(******************************************************************************
Baustein: FB_UnitTestBase
Spezifikation: doc/Spezifikation.pdf, Kap. x.y.z
-------------------------------------------------------------------------------
erstellt:
von:
Geändert:
von:
-------------------------------------------------------------------------------
Beschreibung
Dieser Baustein stellt die Basis für einen Unittest dar und enthält
alle notwendigen Variablen und Methoden zur Testauswertung.

-------------------------------------------------------------------------------
Input
-

Output
	o_eState : EState_t;
	o_eResult: EResult_t;
******************************************************************************)
FUNCTION_BLOCK FB_UnitTestBase
VAR_INPUT
END_VAR
VAR_OUTPUT
	o_eState : EState_t;
	o_eResult: EResult_t;
END_VAR
VAR
	strId	  		: ObjectId_t;
	strClassName	: ObjectId_t;
	strPath			: ObjectId_t;
	strMessage 	 	: StrMessage_t;
	bSkipTest		: BOOL;
	pTestSuite      : TestSuiteHandle_t;
	bRegistered 	: BOOL;
	u32Passed 		: UDINT;
	u32Failed 		: UDINT;
	u32StartTime	: UDINT;
	u32EndTime		: UDINT;
END_VAR

(******************************************************************************
Baustein: FB_UnitTestBase.cleanup
Spezifikation: doc/Spezifikation.pdf, Kap. x.y.z
-------------------------------------------------------------------------------
erstellt:
von:
Geändert:
von:
-------------------------------------------------------------------------------
Beschreibung
Diese Methode...

-------------------------------------------------------------------------------
Input
-

Output
-
******************************************************************************)
{attribute 'hide'} 
METHOD INTERNAL _cleanup : BOOL
VAR_INPUT
END_VAR


	_cleanup := cleanup();
END_METHOD

(******************************************************************************
Baustein: FB_UnitTestBase.execute
Spezifikation: doc/Spezifikation.pdf, Kap. x.y.z
-------------------------------------------------------------------------------
erstellt:
von:
Geändert:
von:
-------------------------------------------------------------------------------
Beschreibung
Diese Methode...

-------------------------------------------------------------------------------
Input
-

Output
-
******************************************************************************)
{attribute 'hide'} 
METHOD INTERNAL _execute : BOOL
VAR_INPUT
END_VAR

	_execute := execute();
END_METHOD

(******************************************************************************
Baustein: FB_UnitTestBase.prepare
Spezifikation: doc/Spezifikation.pdf, Kap. x.y.z
-------------------------------------------------------------------------------
erstellt:
von:
Geändert:
von:
-------------------------------------------------------------------------------
Beschreibung
Diese Methode...

-------------------------------------------------------------------------------
Input
-

Output
-
******************************************************************************)
{attribute 'hide'} 
METHOD INTERNAL _prepare : BOOL
VAR_INPUT
END_VAR

	u32Passed 		:= 0;
	u32Failed 		:= 0;
	u32StartTime 	:= 0;
	u32EndTime 		:= 0;
	o_eResult 		:= EResult_t.eStateSkipped;

	_prepare := prepare();
END_METHOD

(******************************************************************************
Baustein: FB_UnitTestBase.addFailed
Spezifikation: doc/Spezifikation.pdf, Kap. x.y.z
-------------------------------------------------------------------------------
erstellt:
von:
Geändert:
von:
-------------------------------------------------------------------------------
Beschreibung
Diese Methode

-------------------------------------------------------------------------------
Input
-

Output
-
******************************************************************************)
{attribute 'hide'} 
METHOD INTERNAL addFailed : BOOL
VAR_INPUT
	bFatal : BOOL;
END_VAR

	u32Failed := u32Failed + 1;
	
	o_eResult := EResult_t.eStateFailed;
	
	IF bFatal = true THEN
		o_eResult := EResult_t.eStateFailedFatal;
		logError(concat('Test Failed Fatal: ', strId));
	ELSE
		logError(concat('Test Failed : ', strId));
	END_IF
END_METHOD

(******************************************************************************
Baustein: FB_UnitTestBase.addPassed
Spezifikation: doc/Spezifikation.pdf, Kap. x.y.z
-------------------------------------------------------------------------------
erstellt:
von:
Geändert:
von:
-------------------------------------------------------------------------------
Beschreibung
Diese Methode

-------------------------------------------------------------------------------
Input
-

Output
-
******************************************************************************)
{attribute 'hide'} 
METHOD INTERNAL addPassed : BOOL
VAR_INPUT
END_VAR

	u32Passed := u32Passed + 1;

	IF o_eResult = eResult_t.eStateSkipped THEN
		o_eResult := eResult_t.eStatePassed;
	END_IF;
END_METHOD

(******************************************************************************
Baustein: FB_UnitTestBase.assertEQUAL
Spezifikation: doc/Spezifikation.pdf, Kap. x.y.z
-------------------------------------------------------------------------------
erstellt:
von:
Geändert:
von:
-------------------------------------------------------------------------------
Beschreibung
Diese Methode

-------------------------------------------------------------------------------
Input
	Actual   : ANY;
	Expected : ANY;

Output
-
******************************************************************************)
METHOD PROTECTED assertEQUAL : BOOL
VAR_INPUT
	Actual   : ANY;
	Expected : ANY;
END_VAR

	assertEQUAL := FALSE;
	
	IF validate(Actual, Expected) = FALSE THEN
		addFailed(true);
		RETURN;
	END_IF
	
	assertTrue(MEMCMP(Actual.pValue, Expected.pValue, TO_UDINT(Actual.diSize)) = 0);
END_METHOD

(******************************************************************************
Baustein: FB_UnitTestBase.assertEQUAL_Fatal
Spezifikation: doc/Spezifikation.pdf, Kap. x.y.z
-------------------------------------------------------------------------------
erstellt:
von:
Geändert:
von:
-------------------------------------------------------------------------------
Beschreibung
Diese Methode

-------------------------------------------------------------------------------
Input
	Actual   : ANY;
	Expected : ANY;

Output
-
******************************************************************************)
METHOD PROTECTED assertEQUAL_Fatal : BOOL
VAR_INPUT
	Actual   : ANY;
	Expected : ANY;
END_VAR

	assertEQUAL_Fatal := FALSE;
	
	IF validate(Actual, Expected) = FALSE THEN
		addFailed(true);
		RETURN;
	END_IF

	assertTrue_Fatal(MEMCMP(Actual.pValue, Expected.pValue, TO_UDINT(Actual.diSize)) = 0);
END_METHOD

(******************************************************************************
Baustein: FB_UnitTestBase.assertFALSE
Spezifikation: doc/Spezifikation.pdf, Kap. x.y.z
-------------------------------------------------------------------------------
erstellt:
von:
Geändert:
von:
-------------------------------------------------------------------------------
Beschreibung
Diese Methode...

-------------------------------------------------------------------------------
Input
	bValue : BOOL;

Output
-
******************************************************************************)
METHOD PROTECTED assertFALSE : BOOL
VAR_INPUT
	bValue : BOOL;
END_VAR

	IF bValue = FALSE THEN
		addPassed();
	ELSE
		addFailed(bFatal := FALSE);
	END_IF
END_METHOD

(******************************************************************************
Baustein: FB_UnitTestBase.assertFALSE_Fatal
Spezifikation: doc/Spezifikation.pdf, Kap. x.y.z
-------------------------------------------------------------------------------
erstellt:
von:
Geändert:
von:
-------------------------------------------------------------------------------
Beschreibung
Diese Methode

-------------------------------------------------------------------------------
Input
	bValue : BOOL;

Output
-
******************************************************************************)
METHOD PROTECTED assertFALSE_Fatal : BOOL
VAR_INPUT
	bValue : BOOL;
END_VAR

	IF bValue = FALSE THEN
		addPassed();
	ELSE
		addFailed(bFatal := true);
	END_IF
END_METHOD

(******************************************************************************
Baustein: FB_UnitTestBase.assertNotEqual
Spezifikation: doc/Spezifikation.pdf, Kap. x.y.z
-------------------------------------------------------------------------------
erstellt:
von:
Geändert:
von:
-------------------------------------------------------------------------------
Beschreibung
Diese Methode

-------------------------------------------------------------------------------
Input
	Actual   : ANY;
	Expected : ANY;

Output
-
******************************************************************************)
METHOD PROTECTED assertNotEqual : BOOL
VAR_INPUT
	Actual   : ANY;
	Expected : ANY;
END_VAR

	assertNotEqual := FALSE;
	
	IF validate(Actual, Expected) = FALSE THEN
		addFailed(true);
		RETURN;
	END_IF
	
	assertTrue(MEMCMP(Actual.pValue, Expected.pValue, TO_UDINT(Actual.diSize)) <> 0);
END_METHOD

(******************************************************************************
Baustein: FB_UnitTestBase.assertNotEqual_Fatal
Spezifikation: doc/Spezifikation.pdf, Kap. x.y.z
-------------------------------------------------------------------------------
erstellt:
von:
Geändert:
von:
-------------------------------------------------------------------------------
Beschreibung
Diese Methode

-------------------------------------------------------------------------------
Input
	Actual   : ANY;
	Expected : ANY;

Output
-
******************************************************************************)
METHOD PROTECTED assertNotEqual_Fatal : BOOL
VAR_INPUT
	Actual   : ANY;
	Expected : ANY;
END_VAR

	assertNotEqual_Fatal := FALSE;
	
	IF validate(Actual, Expected) = FALSE THEN
		addFailed(true);
		RETURN;
	END_IF
	
	assertTrue_Fatal(MEMCMP(Actual.pValue, Expected.pValue, TO_UDINT(Actual.diSize)) <> 0);
END_METHOD

(******************************************************************************
Baustein: FB_UnitTestBase.assertPtrEqual
Spezifikation: doc/Spezifikation.pdf, Kap. x.y.z
-------------------------------------------------------------------------------
erstellt:
von:
Geändert:
von:
-------------------------------------------------------------------------------
Beschreibung
Diese Methode

-------------------------------------------------------------------------------
Input
	pActual   : PVOID;
	pExpected : PVOID;
	
Output
-
******************************************************************************)
METHOD PROTECTED assertPtrEqual : BOOL
VAR_INPUT
	pActual   : PVOID;
	pExpected : PVOID;
END_VAR

	assertTRUE(pActual = pExpected);
END_METHOD

(******************************************************************************
Baustein: FB_UnitTestBase.assertPtrEqual_Fatal
Spezifikation: doc/Spezifikation.pdf, Kap. x.y.z
-------------------------------------------------------------------------------
erstellt:
von:
Geändert:
von:
-------------------------------------------------------------------------------
Beschreibung
Diese Methode

-------------------------------------------------------------------------------
Input
	pActual   : PVOID;
	pExpected : PVOID;

Output
-
******************************************************************************)
METHOD PROTECTED assertPtrEqual_Fatal : BOOL
VAR_INPUT
	pActual   : PVOID;
	pExpected : PVOID;
END_VAR

	assertTRUE_Fatal(pActual = pExpected);
END_METHOD

(******************************************************************************
Baustein: FB_UnitTestBase.assertPtrNotEqual
Spezifikation: doc/Spezifikation.pdf, Kap. x.y.z
-------------------------------------------------------------------------------
erstellt:
von:
Geändert:
von:
-------------------------------------------------------------------------------
Beschreibung
Diese Methode

-------------------------------------------------------------------------------
Input
	pActual   : PVOID;
	pExpected : PVOID;

Output
-
******************************************************************************)
METHOD PROTECTED assertPtrNotEqual : BOOL
VAR_INPUT
	pActual   : PVOID;
	pExpected : PVOID;
END_VAR

	assertTRUE(pActual <> pExpected);
END_METHOD

(******************************************************************************
Baustein: FB_UnitTestBase.assertPtrNotEqual_Fatal
Spezifikation: doc/Spezifikation.pdf, Kap. x.y.z
-------------------------------------------------------------------------------
erstellt:
von:
Geändert:
von:
-------------------------------------------------------------------------------
Beschreibung
Diese Methode

-------------------------------------------------------------------------------
Input
	pActual   : PVOID;
	pExpected : PVOID;

Output
-
******************************************************************************)
METHOD PROTECTED assertPtrNotEqual_Fatal : BOOL
VAR_INPUT
	pActual   : PVOID;
	pExpected : PVOID;
END_VAR

	assertTRUE_Fatal(pActual <> pExpected);
END_METHOD

(******************************************************************************
Baustein: FB_UnitTestBase.assertPtrNotNull
Spezifikation: doc/Spezifikation.pdf, Kap. x.y.z
-------------------------------------------------------------------------------
erstellt:
von:
Geändert:
von:
-------------------------------------------------------------------------------
Beschreibung
Diese Methode

-------------------------------------------------------------------------------
Input
	pActual   : PVOID;

Output
-
******************************************************************************)
METHOD PROTECTED assertPtrNotNull : BOOL
VAR_INPUT
	pActual   : PVOID;
END_VAR

	assertTRUE(pActual <> 0);
END_METHOD

(******************************************************************************
Baustein: FB_UnitTestBase.assertPtrNotNull_Fatal
Spezifikation: doc/Spezifikation.pdf, Kap. x.y.z
-------------------------------------------------------------------------------
erstellt:
von:
Geändert:
von:
-------------------------------------------------------------------------------
Beschreibung
Diese Methode

-------------------------------------------------------------------------------
Input
	pActual   : PVOID;

Output
-
******************************************************************************)
METHOD PROTECTED assertPtrNotNull_Fatal : BOOL
VAR_INPUT
	pActual   : PVOID;
END_VAR

	assertTRUE_Fatal(pActual <> 0);
END_METHOD

(******************************************************************************
Baustein: FB_UnitTestBase.assertPtrNull
Spezifikation: doc/Spezifikation.pdf, Kap. x.y.z
-------------------------------------------------------------------------------
erstellt:
von:
Geändert:
von:
-------------------------------------------------------------------------------
Beschreibung
Diese Methode

-------------------------------------------------------------------------------
Input
	pActual   : PVOID;

Output
-
******************************************************************************)
METHOD PROTECTED assertPtrNull : BOOL
VAR_INPUT
	pActual   : PVOID;
END_VAR

	assertTRUE(pActual = 0);
END_METHOD

(******************************************************************************
Baustein: FB_UnitTestBase.assertPtrNull_Fatal
Spezifikation: doc/Spezifikation.pdf, Kap. x.y.z
-------------------------------------------------------------------------------
erstellt:
von:
Geändert:
von:
-------------------------------------------------------------------------------
Beschreibung
Diese Methode

-------------------------------------------------------------------------------
Input
	pActual   : PVOID;

Output
-
******************************************************************************)
METHOD PROTECTED assertPtrNull_Fatal : BOOL
VAR_INPUT
	pActual   : PVOID;
END_VAR

	assertTRUE_Fatal(pActual = 0);
END_METHOD

(******************************************************************************
Baustein: FB_UnitTestBase.assertRealEqual
Spezifikation: doc/Spezifikation.pdf, Kap. x.y.z
-------------------------------------------------------------------------------
erstellt:
von:
Geändert:
von:
-------------------------------------------------------------------------------
Beschreibung
Diese Methode

-------------------------------------------------------------------------------
Input
	r32Actual 		: REAL;
	r32Expected 	: REAL;
	r32Granularity 	: REAL;

Output
-
******************************************************************************)
METHOD PROTECTED assertRealEqual : BOOL
VAR_INPUT
	r32Actual 		: REAL;
	r32Expected 	: REAL;
	r32Granularity 	: REAL;
END_VAR

	assertTRUE(ABS(r32Actual-r32Expected) <= ABS(r32Granularity));
END_METHOD

(******************************************************************************
Baustein: FB_UnitTestBase.assertRealEqual_Fatal
Spezifikation: doc/Spezifikation.pdf, Kap. x.y.z
-------------------------------------------------------------------------------
erstellt:
von:
Geändert:
von:
-------------------------------------------------------------------------------
Beschreibung
Diese Methode

-------------------------------------------------------------------------------
Input
	r32Actual 		: REAL;
	r32Expected 	: REAL;
	r32Granularity 	: REAL;

Output
-
******************************************************************************)
METHOD PROTECTED assertRealEqual_Fatal : BOOL
VAR_INPUT
	r32Actual 		: REAL;
	r32Expected 	: REAL;
	r32Granularity 	: REAL;
END_VAR

	assertTRUE_Fatal(ABS(r32Actual-r32Expected) <= ABS(r32Granularity));
END_METHOD

(******************************************************************************
Baustein: FB_UnitTestBase.assertRealNotEqual
Spezifikation: doc/Spezifikation.pdf, Kap. x.y.z
-------------------------------------------------------------------------------
erstellt:
von:
Geändert:
von:
-------------------------------------------------------------------------------
Beschreibung
Diese Methode

-------------------------------------------------------------------------------
Input
	r32Actual 		: REAL;
	r32Expected 	: REAL;
	r32Granularity 	: REAL;

Output
-
******************************************************************************)
METHOD PRIVATE assertRealNotEqual : BOOL
VAR_INPUT
	r32Actual 		: REAL;
	r32Expected 	: REAL;
	r32Granularity 	: REAL;
END_VAR

	assertTRUE(ABS(r32Actual-r32Expected) > ABS(r32Granularity));
END_METHOD

(******************************************************************************
Baustein: FB_UnitTestBase.assertRealNotEqual_Fatal
Spezifikation: doc/Spezifikation.pdf, Kap. x.y.z
-------------------------------------------------------------------------------
erstellt:
von:
Geändert:
von:
-------------------------------------------------------------------------------
Beschreibung
Diese Methode

-------------------------------------------------------------------------------
Input
	r32Actual 		: REAL;
	r32Expected 	: REAL;
	r32Granularity 	: REAL;

Output
-
******************************************************************************)
METHOD PROTECTED assertRealNotEqual_Fatal : BOOL
VAR_INPUT
	r32Actual 		: REAL;
	r32Expected 	: REAL;
	r32Granularity 	: REAL;
END_VAR

	assertTRUE_Fatal(ABS(r32Actual-r32Expected) > ABS(r32Granularity));
END_METHOD

(******************************************************************************
Baustein: FB_UnitTestBase.assertStringEqual
Spezifikation: doc/Spezifikation.pdf, Kap. x.y.z
-------------------------------------------------------------------------------
erstellt:
von:
Geändert:
von:
-------------------------------------------------------------------------------
Beschreibung
Diese Methode

-------------------------------------------------------------------------------
Input
	pActual 	: StringHandle_t;
	pExpected 	: StringHandle_t;

Output
-
******************************************************************************)
METHOD PROTECTED assertStringEqual : BOOL
VAR_INPUT
	pActual 	: StringHandle_t;
	pExpected 	: StringHandle_t;
END_VAR

	IF strncmp(pActual, pExpected, LEN(pExpected^)) = TRUE THEN
		addPassed();
	ELSE
		addFailed(bFatal := FALSE);		
	END_IF
END_METHOD

(******************************************************************************
Baustein: FB_UnitTestBase.assertStringEqual_Fatal
Spezifikation: doc/Spezifikation.pdf, Kap. x.y.z
-------------------------------------------------------------------------------
erstellt:
von:
Geändert:
von:
-------------------------------------------------------------------------------
Beschreibung
Diese Methode

-------------------------------------------------------------------------------
Input
	pActual 	: StringHandle_t;
	pExpected 	: StringHandle_t;

Output
-
******************************************************************************)
METHOD PROTECTED assertStringEqual_Fatal : BOOL
VAR_INPUT
	pActual 	: StringHandle_t;
	pExpected 	: StringHandle_t;
END_VAR

	IF strncmp(pActual, pExpected, LEN(pExpected^)) = TRUE THEN
		addPassed();
	ELSE
		addFailed(bFatal := TRUE);		
	END_IF
END_METHOD

(******************************************************************************
Baustein: FB_UnitTestBase.assertStringNotEqual
Spezifikation: doc/Spezifikation.pdf, Kap. x.y.z
-------------------------------------------------------------------------------
erstellt:
von:
Geändert:
von:
-------------------------------------------------------------------------------
Beschreibung
Diese Methode

-------------------------------------------------------------------------------
Input
	pActual 	: StringHandle_t;
	pExpected 	: StringHandle_t;

Output
-
******************************************************************************)
METHOD PROTECTED assertStringNotEqual : BOOL
VAR_INPUT
	pActual 	: StringHandle_t;
	pExpected 	: StringHandle_t;
END_VAR

	IF strncmp(pActual, pExpected, LEN(pExpected^)) = false THEN
		addPassed();
	ELSE
		addFailed(bFatal := FALSE);		
	END_IF
END_METHOD

(******************************************************************************
Baustein: FB_UnitTestBase.assertStringNotEqual_fatal
Spezifikation: doc/Spezifikation.pdf, Kap. x.y.z
-------------------------------------------------------------------------------
erstellt:
von:
Geändert:
von:
-------------------------------------------------------------------------------
Beschreibung
Diese Methode

-------------------------------------------------------------------------------
Input
	pExpected 	: StringHandle_t;
	pActual 	: StringHandle_t;

Output
-
******************************************************************************)
METHOD PROTECTED assertStringNotEqual_fatal : BOOL
VAR_INPUT
	pExpected 	: StringHandle_t;
	pActual 	: StringHandle_t;
END_VAR

	IF strncmp(pActual, pExpected, LEN(pExpected^)) = FALSE THEN
		addPassed();
	ELSE
		addFailed(bFatal := TRUE);		
	END_IF
END_METHOD

(******************************************************************************
Baustein: FB_UnitTestBase.assertTRUE
Spezifikation: doc/Spezifikation.pdf, Kap. x.y.z
-------------------------------------------------------------------------------
erstellt:
von:
Geändert:
von:
-------------------------------------------------------------------------------
Beschreibung
Diese Methode...

-------------------------------------------------------------------------------
Input
	bValue : BOOL;

Output
-
******************************************************************************)
METHOD PROTECTED assertTRUE : BOOL
VAR_INPUT
	bValue : BOOL;
END_VAR

	IF bValue = true THEN
		addPassed();
	ELSE
		addFailed(bFatal := FALSE);
	END_IF
END_METHOD


(******************************************************************************
Baustein: FB_UnitTestBase.assertTRUE_Fatal
Spezifikation: doc/Spezifikation.pdf, Kap. x.y.z
-------------------------------------------------------------------------------
erstellt:
von:
Geändert:
von:
-------------------------------------------------------------------------------
Beschreibung
Diese Methode

-------------------------------------------------------------------------------
Input
-

Output
-
******************************************************************************)
METHOD PROTECTED assertTRUE_Fatal : BOOL
VAR_INPUT
	bValue : BOOL;
END_VAR

	IF bValue = TRUE THEN
		addPassed();
	ELSE
		addFailed(bFatal := true);
	END_IF
END_METHOD

(******************************************************************************
Baustein: FB_UnitTestBase.cleanup
Spezifikation: doc/Spezifikation.pdf, Kap. x.y.z
-------------------------------------------------------------------------------
erstellt:
von:
Geändert:
von:
-------------------------------------------------------------------------------
Beschreibung
Diese Methode...

-------------------------------------------------------------------------------
Input
-

Output
-
******************************************************************************)
METHOD PUBLIC cleanup : BOOL
VAR_INPUT
END_VAR


	cleanup := false;
END_METHOD

(******************************************************************************
Baustein: FB_UnitTestBase.execute
Spezifikation: doc/Spezifikation.pdf, Kap. x.y.z
-------------------------------------------------------------------------------
erstellt:
von:
Geändert:
von:
-------------------------------------------------------------------------------
Beschreibung
Diese Methode...

-------------------------------------------------------------------------------
Input
-

Output
-
******************************************************************************)
METHOD PUBLIC execute : BOOL
VAR_INPUT
END_VAR

	Execute := false;
END_METHOD

(******************************************************************************
Baustein: FB_Testsuite.FB_init
Spezifikation: doc/Spezifikation.pdf, Kap. x.y.z
-------------------------------------------------------------------------------
erstellt:
von:
Geändert:
von:
-------------------------------------------------------------------------------
Beschreibung
Diese Methode

-------------------------------------------------------------------------------
Input
-

Output
-
******************************************************************************)
{attribute 'hide'} 
METHOD FB_init : BOOL
VAR_INPUT
	bInitRetains 	: BOOL; // if TRUE, the retain variables are initialized (warm start / cold start)
	bInCopyCode 	: BOOL;  // if TRUE, the instance afterwards gets moved into the copy code (online change)
	i_strId	  		: ObjectId_t;
	i_strClassName	: ObjectId_t;
	i_strPath 		: ObjectId_t;
	i_pTestSuite 	: TestSuiteHandle_t;
	i_bExecute      : BOOL := true; 
END_VAR
	
	strId 		 := i_strId;
	strClassName := i_strClassName;
	strPath 	 := i_strPath;
	bSkipTest  	 := (i_bExecute = false);
	pTestSuite 	 := i_pTestSuite;
	
	register();
END_METHOD

(******************************************************************************
Baustein: FB_UnitTestBase.getId
Spezifikation: doc/Spezifikation.pdf, Kap. x.y.z
-------------------------------------------------------------------------------
erstellt:
von:
Geändert:
von:
-------------------------------------------------------------------------------
Beschreibung
Diese Methode

-------------------------------------------------------------------------------
Input
-

Output
-
******************************************************************************)
{attribute 'hide'} 
METHOD PUBLIC getClassName : ObjectId_t
VAR_INPUT
END_VAR

	getClassName := strClassName;
END_METHOD

(******************************************************************************
Baustein: FB_UnitTestBase.getFailed
Spezifikation: doc/Spezifikation.pdf, Kap. x.y.z
-------------------------------------------------------------------------------
erstellt:
von:
Geändert:
von:
-------------------------------------------------------------------------------
Beschreibung
Diese Methode

-------------------------------------------------------------------------------
Input
-

Output
-
******************************************************************************)
{attribute 'hide'} 
METHOD PUBLIC getFailed : UDINT
VAR_INPUT
END_VAR

	getFailed := u32Failed;
END_METHOD

(******************************************************************************
Baustein: FB_UnitTestBase.getId
Spezifikation: doc/Spezifikation.pdf, Kap. x.y.z
-------------------------------------------------------------------------------
erstellt:
von:
Geändert:
von:
-------------------------------------------------------------------------------
Beschreibung
Diese Methode

-------------------------------------------------------------------------------
Input
-

Output
-
******************************************************************************)
{attribute 'hide'} 
METHOD PUBLIC getId : ObjectId_t
VAR_INPUT
END_VAR

	getId := strId;
END_METHOD

METHOD PUBLIC getMessage : StrMessage_t
VAR_INPUT
END_VAR

	getMessage := strMessage;
END_METHOD

(******************************************************************************
Baustein: FB_UnitTestBase.getPassed
Spezifikation: doc/Spezifikation.pdf, Kap. x.y.z
-------------------------------------------------------------------------------
erstellt:
von:
Geändert:
von:
-------------------------------------------------------------------------------
Beschreibung
Diese Methode

-------------------------------------------------------------------------------
Input
-

Output
-
******************************************************************************)
{attribute 'hide'} 
METHOD PUBLIC getPassed : UDINT
VAR_INPUT
END_VAR

	getPassed := u32Passed;
END_METHOD

(******************************************************************************
Baustein: FB_UnitTestBase.getPassed
Spezifikation: doc/Spezifikation.pdf, Kap. x.y.z
-------------------------------------------------------------------------------
erstellt:
von:
Geändert:
von:
-------------------------------------------------------------------------------
Beschreibung
Diese Methode

-------------------------------------------------------------------------------
Input
-

Output
-
******************************************************************************)
{attribute 'hide'} 
METHOD PUBLIC getPath : ObjectId_t
VAR_INPUT
END_VAR

	getPath := strPath;
END_METHOD

(******************************************************************************
Baustein: FB_UnitTestBase.getPassed
Spezifikation: doc/Spezifikation.pdf, Kap. x.y.z
-------------------------------------------------------------------------------
erstellt:
von:
Geändert:
von:
-------------------------------------------------------------------------------
Beschreibung
Diese Methode

-------------------------------------------------------------------------------
Input
-

Output
-
******************************************************************************)
{attribute 'hide'} 
METHOD PRIVATE getSystemTime : UDINT
VAR_INPUT
END_VAR
VAR
	u64Time : ULINT;
END_VAR

	u64Time := F_GetSystemTime()/10000;


	getSystemTime := to_udint(u64Time and 16#FFFFFFFF);
END_METHOD

(******************************************************************************
Baustein: FB_UnitTestBase.getPassed
Spezifikation: doc/Spezifikation.pdf, Kap. x.y.z
-------------------------------------------------------------------------------
erstellt:
von:
Geändert:
von:
-------------------------------------------------------------------------------
Beschreibung
Diese Methode

-------------------------------------------------------------------------------
Input
-

Output
-
******************************************************************************)
{attribute 'hide'} 
METHOD PUBLIC getTime : UDINT
VAR_INPUT
END_VAR

	getTime := 0;

	IF u32EndTime > u32StartTime THEN
		getTime := u32EndTime - u32StartTime;
	END_IF;
END_METHOD

(******************************************************************************
Baustein: FB_UnitTestBase.getPassed
Spezifikation: doc/Spezifikation.pdf, Kap. x.y.z
-------------------------------------------------------------------------------
erstellt:
von:
Geändert:
von:
-------------------------------------------------------------------------------
Beschreibung
Diese Methode

-------------------------------------------------------------------------------
Input
-

Output
-
******************************************************************************)
{attribute 'hide'} 
METHOD INTERNAL isSkipped : BOOL
VAR_INPUT
END_VAR

	isSkipped := bSkipTest;
END_METHOD

(******************************************************************************
Baustein: FB_UnitTestBase.logError
Spezifikation: doc/Spezifikation.pdf, Kap. x.y.z
-------------------------------------------------------------------------------
erstellt:
von:
Geändert:
von:
-------------------------------------------------------------------------------
Beschreibung
Diese Methode

-------------------------------------------------------------------------------
Input
-

Output
-
******************************************************************************)
{attribute 'hide'} 
METHOD PROTECTED logError : BOOL
VAR_INPUT
	i_strMessage : StrMessage_t;
END_VAR

	ADSLOGSTR(msgCtrlMask 	:= ADSLOG_MSGTYPE_ERROR , 
			  msgFmtStr 	:= i_strMessage, 
			  strArg 		:= '');
END_METHOD

(******************************************************************************
Baustein: FB_UnitTestBase.logInfo
Spezifikation: doc/Spezifikation.pdf, Kap. x.y.z
-------------------------------------------------------------------------------
erstellt:
von:
Geändert:
von:
-------------------------------------------------------------------------------
Beschreibung
Diese Methode

-------------------------------------------------------------------------------
Input
-

Output
-
******************************************************************************)
{attribute 'hide'} 
METHOD INTERNAL logInfo : BOOL
VAR_INPUT
	i_strMessage : StrMessage_t;
END_VAR

	ADSLOGSTR(msgCtrlMask 	:= ADSLOG_MSGTYPE_HINT , 
			  msgFmtStr 	:= i_strMessage, 
			  strArg 		:= '');
END_METHOD

(******************************************************************************
Baustein: FB_UnitTestBase.prepare
Spezifikation: doc/Spezifikation.pdf, Kap. x.y.z
-------------------------------------------------------------------------------
erstellt:
von:
Geändert:
von:
-------------------------------------------------------------------------------
Beschreibung
Diese Methode...

-------------------------------------------------------------------------------
Input
-

Output
-
******************************************************************************)
METHOD PUBLIC prepare : BOOL
VAR_INPUT
END_VAR

	prepare := false;
END_METHOD

(******************************************************************************
Baustein: FB_UnitTestBase.register
Spezifikation: doc/Spezifikation.pdf, Kap. x.y.z
-------------------------------------------------------------------------------
erstellt:
von:
Geändert:
von:
-------------------------------------------------------------------------------
Beschreibung
Diese Methode

-------------------------------------------------------------------------------
Input
-

Output
-
******************************************************************************)
{attribute 'hide'} 
METHOD INTERNAL register : BOOL
VAR_INPUT
END_VAR

	IF pTestSuite <> 0 	AND 
       bRegistered = FALSE  THEN
		
		bRegistered := pTestSuite^.addTestcase(THIS);
	
	END_IF
END_METHOD

(******************************************************************************
Baustein: FB_UnitTestBase.getPassed
Spezifikation: doc/Spezifikation.pdf, Kap. x.y.z
-------------------------------------------------------------------------------
erstellt:
von:
Geändert:
von:
-------------------------------------------------------------------------------
Beschreibung
Diese Methode

-------------------------------------------------------------------------------
Input
-

Output
-
******************************************************************************)
{attribute 'hide'} 
METHOD INTERNAL setEndTime : BOOL
VAR_INPUT
END_VAR

	IF u32EndTime = 0 THEN
		u32EndTime := getSystemTime();
	END_IF;
	setEndTime := true;
END_METHOD

METHOD PROTECTED setMessage
VAR_INPUT
	strValue : StrMessage_t;
END_VAR

	IF o_eResult < EResult_t.eStateFailed THEN
		strMessage := strValue;
	END_IF;
END_METHOD

(******************************************************************************
Baustein: FB_UnitTestBase.getPassed
Spezifikation: doc/Spezifikation.pdf, Kap. x.y.z
-------------------------------------------------------------------------------
erstellt:
von:
Geändert:
von:
-------------------------------------------------------------------------------
Beschreibung
Diese Methode

-------------------------------------------------------------------------------
Input
-

Output
-
******************************************************************************)
{attribute 'hide'} 
METHOD INTERNAL setStartTime : BOOL
VAR_INPUT
END_VAR

	IF u32StartTime = 0 THEN
		u32StartTime   	:= getSystemTime();
	END_IF;
	setStartTime := true;
END_METHOD

(******************************************************************************
Baustein: FB_UnitTestBase.strncmp
Spezifikation: doc/Spezifikation.pdf, Kap. x.y.z
-------------------------------------------------------------------------------
erstellt:
von:
Geändert:
von:
-------------------------------------------------------------------------------
Beschreibung
Diese Methode

-------------------------------------------------------------------------------
Input
	strInput 	: StringHandle_t;
	strCompare 	: StringHandle_t;
	s16Size		: INT;

Output
-
******************************************************************************)
{attribute 'hide'} 
METHOD PRIVATE strncmp : BOOL
VAR_INPUT
	strInput 	: StringHandle_t;
	strCompare 	: StringHandle_t;
	s16Size		: INT;
END_VAR
VAR
	s16Size1 : INT;
	s16Size2 : INT;
	s16Diff  : INT;
END_VAR

   s16Size1:= LEN(strInput^); 
	s16Size2:= LEN(strCompare^); 
	
	strncmp := FALSE;
	
	s16Diff := s16Size1 - s16Size2;
   
	// vergleich nur wenn beide Strings
	// gleich groß sind.
	IF s16Diff  = 0 THEN

		strncmp := TRUE;
	
		WHILE(s16Size > 0) DO

			IF strInput^ <> strCompare^ THEN
				strncmp := FALSE;
			END_IF;  
 
			strInput   := strInput + 1;
			strCompare := strCompare + 1;
			s16Size    := s16Size - 1;

		END_WHILE


	
	END_IF;
END_METHOD

(******************************************************************************
Baustein: FB_UnitTestBase.validate
Spezifikation: doc/Spezifikation.pdf, Kap. x.y.z
-------------------------------------------------------------------------------
erstellt:
von:
Geändert:
von:
-------------------------------------------------------------------------------
Beschreibung
Diese Methode

-------------------------------------------------------------------------------
Input
	var1 : ANY;
	var2 : ANY;

Output
-
******************************************************************************)
{attribute 'hide'} 
METHOD PRIVATE validate : BOOL
VAR_INPUT
	var1 : ANY;
	var2 : ANY;
END_VAR

	validate := FALSE;
	
	IF (var1.pValue = 0 OR var2.pValue = 0) THEN
		RETURN;
	END_IF

	IF (var1.TypeClass <> var2.TypeClass) THEN
		RETURN;
	END_IF;	
	
	IF (var1.diSize <> var2.diSize) THEN
		RETURN;
	END_IF;	
	
	validate := true;
END_METHOD

END_FUNCTION_BLOCK

(* stored: Version 1.1.0.1, ProductVersion 3.1.4024.6
   POU FB_UnitTestBase: Id {77b52f8d-9a49-403a-aba1-80915f687878}, SpecialFunc None
   Method _cleanup: Id {344aee8e-b817-4cb6-9aba-783306fb7b3f}
   Method _execute: Id {7a2e47ea-4d60-41f0-a3d6-a81f0185c513}
   Method _prepare: Id {542f6515-c2b9-44d6-8c08-2dee2ccb31ed}
   Method addFailed: Id {877265ac-7517-465d-8046-dbd413ab22a9}
   Method addPassed: Id {725a8b74-1eab-4dbd-9f39-193c14d3c944}
   Method assertEQUAL: Id {ad51daad-5695-45d0-ad00-7926bcc015fa}
   Method assertEQUAL_Fatal: Id {69be4dda-87a9-4f6f-9eca-8a1ee02fedac}
   Method assertFALSE: Id {d4d5eea3-3c53-497c-9176-1d2814a51e39}
   Method assertFALSE_Fatal: Id {75476dd2-303d-4781-a584-de30bb3a6473}
   Method assertNotEqual: Id {7bdd8554-52a7-414f-8a4a-343d38a85ee0}
   Method assertNotEqual_Fatal: Id {50f19e45-a9a3-4436-9481-7ad1f66a8015}
   Method assertPtrEqual: Id {95a0bcc0-afe3-4228-85a2-ce212c091a6f}
   Method assertPtrEqual_Fatal: Id {1b8e3907-0f7e-4c04-80e7-103c2b3a23a5}
   Method assertPtrNotEqual: Id {57846629-242c-4e81-af74-58586a21a4fc}
   Method assertPtrNotEqual_Fatal: Id {39a47f2c-67f8-43f2-bc30-f2cb3de76090}
   Method assertPtrNotNull: Id {f628fc0d-4d94-48e7-aae3-588658d79bb7}
   Method assertPtrNotNull_Fatal: Id {02ae7d7d-3ede-4c25-85fd-0879e689222b}
   Method assertPtrNull: Id {abd2bd77-de32-4620-9218-680a260e8028}
   Method assertPtrNull_Fatal: Id {5bf9c97f-bc97-48db-98fa-ba9cb62263a9}
   Method assertRealEqual: Id {d770309a-bad4-4c69-b79f-274b8b36691a}
   Method assertRealEqual_Fatal: Id {cf2c2abf-779b-4ad8-b6e5-676b71c0ac70}
   Method assertRealNotEqual: Id {78d62bc5-9b58-4d56-afb5-189d3abc8861}
   Method assertRealNotEqual_Fatal: Id {258a11aa-40fa-4616-826d-01f5de63c20d}
   Method assertStringEqual: Id {83105799-7b7a-4d3d-8679-14126f120e79}
   Method assertStringEqual_Fatal: Id {bf1be694-6409-4e9e-9292-da4654ce1902}
   Method assertStringNotEqual: Id {5b6c5929-a0bc-40c1-a6e9-53f688e2534b}
   Method assertStringNotEqual_fatal: Id {5f4342ff-8918-48d1-98ef-3f0b434e545d}
   Method assertTRUE: Id {22cc59e3-d507-4b30-a16f-46ddc4d327da}
   Method assertTRUE_Fatal: Id {33bf9cec-0e76-4b31-9c97-1667bb6d5ac6}
   Method cleanup: Id {bb611570-6ab2-451b-9f0d-51e2ce59af0a}
   Method execute: Id {eaaea70b-9bf9-4b40-b05d-957421faa196}
   Method FB_init: Id {4cb36c1a-3bd9-4b40-bdb1-0e89fb27e2fa}
   Method getClassName: Id {fe0c9224-6b8f-4968-bd60-2e0b1dc4c7d8}
   Method getFailed: Id {03b873b5-0f90-4435-8771-5dc65ef5e0d1}
   Method getId: Id {3201004a-c0ba-477e-8045-eedf4c12dcd0}
   Method getMessage: Id {afb1fb13-c5eb-4812-98a0-96deb4f8231a}
   Method getPassed: Id {2d53e756-4b16-44f6-b072-8c9bc39b56a8}
   Method getPath: Id {e3a99e4d-69cf-4522-86d0-57b9b9298cbb}
   Method getSystemTime: Id {dc291d5d-13e7-498d-ab24-a88e76a0f5f2}
   Method getTime: Id {289a6643-aea8-41f4-9573-9f8f1e125c8e}
   Method isSkipped: Id {e2151300-eb3a-4ef7-9340-3371bd55a074}
   Method logError: Id {16a351f0-cd4d-4e8b-bead-0c78616d52ea}
   Method logInfo: Id {2a28e610-d91b-4870-a421-7bc6546ff390}
   Method prepare: Id {571b8d1e-086f-4be7-aee6-f996b70e4b02}
   Method register: Id {4a228bed-2579-4e19-893d-8dcd5cfaa8a3}
   Method setEndTime: Id {2f133e6d-150e-424a-a9c1-5a581e939cfa}
   Method setMessage: Id {5e945eba-6cfb-4739-8a87-efafbad421bc}
   Method setStartTime: Id {8cc3bd6c-8aa2-4c8c-8cf1-b74a81a48cb3}
   Method strncmp: Id {ba3fcb40-c976-48c8-9fd0-cd1feb115e5f}
   Method validate: Id {26cbef17-aced-449e-9fb6-d6b834f5b8ef} *)
